FUNCTION_BLOCK PassiveRoom IMPLEMENTS I_Execute, I_Init
VAR CONSTANT
	STATE_CAP		: UDINT := 5;
END_VAR
VAR
	_this			: Entity;
	_ctx			: Room_Ctx;
	_room			: RoomInterface(_ctx);
	_tag			: Tag(CONCAT('Room_', UDINT_TO_STRING(_room.Id)));
	_compTag		: Comp(_tag, _this);
	_init			: Init(THIS^);
	_exe			: Execute(THIS^);
	
	_uiLogic		: Room_UiLogic(_ctx);
	
	_onSystemEvent	: Room_OnSystemEvent(_ctx);
	
	_smgr			: StateManager<STATE_CAP>(_this);
	_proxSmgr		: StateManagerProxy(_smgr, _ctx.state.iMgr);
	
	_disable		: Room_State_Disabled(_this, _ctx);
	_proxDisable	: StateProxy(_disable, _ctx.state.iDisable);
	
	_fault			: Room_State_Fault(_this,_ctx);
	_proxFault		: StateProxy(_fault, _ctx.state.iFault);	
	
	_idle			: Room_State_Idle(_this,_ctx);
	_proxIdle		: StateProxy(_idle, _ctx.state.iIdle);	
	
	_systemOff		: Room_State_SystemOff(_this,_ctx);
	_proxSystemOff	: StateProxy(_systemOff, _ctx.state.iSystemOff);
END_VAR

// Here add custom components

VAR PERSISTENT
	_bEnablePassive	: BOOL;
END_VAR
VAR_INPUT
	bInletValveIsOpen		: BOOL;
	bInletValveIsClosed		: BOOL;
	
	bOutletValveIsOpen		: BOOL;
	bOutletValveIsClosed	: BOOL;
END_VAR
VAR_OUTPUT
	bInletValve			: BOOL;
	bOutletValve		: BOOL;
END_VAR
VAR
	_passiveDemand	: Room_State_DemandPassive(_this, _ctx, _bEnablePassive);
	
	_simInlet		: ValveSim;
	_simOutlet		: ValveSim;
END_VAR

METHOD Execute
_ctx.priv.bClosed := bInletValveIsClosed AND bOutletValveIsClosed;
_ctx.priv.bOpen := bInletValveIsOpen AND bOutletValveIsOpen;

bInletValve :=  _ctx.io.bOpenValves;
bOutletValve :=  _ctx.io.bOpenValves;

_ctx.hmi.sData := '';

// SIMULATION

_simInlet(bInput := bInletValve,
			bFault := sim.param.bToggleValveFault,
			bIsOpen := bInletValveIsOpen,
			bIsClosed := bInletValveIsClosed);
_simOutlet(bInput := bOutletValve,
			bFault := sim.param.bToggleValveFault,
			bIsOpen := bOutletValveIsOpen,
			bIsClosed := bOutletValveIsClosed);

IF NOT sim.bTick THEN
	RETURN;
END_IF

IF bInletValve AND bOutletValve THEN
	sim.rSystemTemperature := sim.rSystemTemperature + sim.param.rSystemTemperatureDropPerHeater * LREAL_TO_REAL(Random());
END_IF
END_METHOD

METHOD Init
_smgr.Request(_idle);
END_METHOD

END_FUNCTION_BLOCK

(* stored: Version 1.1.0.1
   POU PassiveRoom: Id {6ae55b71-3bf9-4dce-a2da-1a8618e62628}, SpecialFunc None
   Method Execute: Id {6b5be57a-f08a-4fb9-be69-3005ba5b1cc8}
   Method Init: Id {718dfcb2-f799-42f7-832b-c159fdd31449} *)
